TYPE ST_CommunicationMetaData :
STRUCT
	cbLen	: UDINT;
	pData	: PVOID;
END_STRUCT
END_TYPE

(* stored: Version 1.1.0.1, ProductVersion 3.1.4024.15
   DUT ST_CommunicationMetaData: Id {fdcf7125-81a2-4c5f-88ad-e865feb496c5} *)
